FUNCTION F_GetDestination : ST_PositionIdent
(**************************************************************************************
 * 	Application		:	BoxControl Framework
 *	Revision		:	$Revision: 404529 $
 *	Revision date	:	$Date: 2018-04-23 08:21:38 +0200 (Mo., 23 Apr 2018) $
 *	Last changed by	:	$Author: b7bolm $
 *	URL				:	$URL: http://almscdc.swisslog.com/repo/SWPD/Development/BoxControlFramework/20_Release/trunk/01_Software/BCF/BCF/JumpStart/20_Product/10_App/12_E_Functions/10_Lib/10_Conv/10_Functions/F_GetDestination.TcPOU $
 *
 *	Purpose			:	Gets the specified destination of a position
 *
 * ------------------------------------------------------------------------------------
 *	Copyright Swisslog [IP AG], Switzerland. All rights reserved.
 * 
 * ------------------------------------------------------------------------------------
 *	
 * 	Revision History: 
 *
 * 	VERSION			DATE			INITIALS			DESCRIPTION
 *	0.1				01.01.2001		swl					Example
 *
 **************************************************************************************)
VAR_INPUT
	eFunctionNumber		: E_FunctionNumber; // Function number
	ZoneNumber			: INT; // ZoneNumber
	DestinationIdx		: INT; // Which destination slot (Default 1)
END_VAR

VAR
	TU_DataIndex		: DINT;
END_VAR

// Init
F_GetDestination.eFunctionNumber := E_FunctionNumber.F_BEGIN_FUNCTION;
F_GetDestination.ZoneNumber	:= 0;

// Validate inputs
IF eFunctionNumber > E_FunctionNumber.F_BEGIN_FUNCTION AND
   eFunctionNumber < E_FunctionNumber.F_END_FUNCTION AND
   ZoneNumber > 0 AND
   ZoneNumber <= Conveyor.NUMBER_OF_ZONES_PER_FUNCTION THEN
   	// If zone is valid and consists of a TU-Data index
	IF __ISVALIDREF(FunctionRegistry[eFunctionNumber].Zone[ZoneNumber].refZoneData) THEN
		TU_DataIndex := FunctionRegistry[eFunctionNumber].Zone[ZoneNumber].refZoneData.TransportControlData.TU_DataIndex;
		// Return destination slot
		IF DestinationIdx > 0 AND DestinationIdx <= Conveyor.NUMBER_OF_DESTINATIONS THEN
			F_GetDestination.eFunctionNumber := TU_DataTable[TU_DataIndex].Destination[DestinationIdx].eFunctionNumber;
			F_GetDestination.ZoneNumber	:= TU_DataTable[TU_DataIndex].Destination[DestinationIdx].ZoneNumber;;
		END_IF
	END_IF
END_IF

END_FUNCTION

(* stored: Version 1.1.0.1, ProductVersion 3.1.4022.12
   POU F_GetDestination: Id {c58bd7ab-9081-46c6-a91a-7418875d8fd7}, SpecialFunc None *)
